INTERFACE IPAFDischarging EXTENDS IPAProcessFunction

END_INTERFACE

(* stored: Version 1.1.0.1, ProductVersion 3.1.4020.12
   Itf IPAFDischarging: Id {85ea922b-a471-4480-ab70-966f1cfadecb} *)
